{attribute 'Tc2GvlVarNames'}
(* Generated automatically by TwinCAT - (read only) *)
VAR_CONFIG
END_VAR

(* stored: Version 1.1.0.1, ProductVersion 3.1.4022.16
   GVL TwinCAT_Configuration: Id {b8dc3bf4-4caa-45e3-9abc-cd5a914880c4} *)
